FUNCTION_BLOCK FB_WindingControl
VAR_INPUT
	// Input hmi connection from MAIN
	hmiConnection   : POINTER TO FB_hmi_connection;   // HMI connection
	eventLogger     : POINTER TO FB_EventLogger;      // Event logger
	fileReadWrite   : POINTER TO FB_fileReadWrite;    // File read/write
END_VAR

VAR
	// Temporary testing vars

	// Function Blocks

	// CONTROL VARS
	desiredTension          : LREAL := 0;         // Desired tension
	desiredLinspeed         : LREAL := 0;         // Desired linear speed
	unwinding               : BOOL  := FALSE;     // Unwinding flag
	desiredTurnCountPickup  : DINT  := 0;         // Desired turn count for pickup
	
	// Exit conditions
	target_turn_count       : DINT  := 0;         // Target turn count

	// STATUS VARS
	state                   : INT   := 0;         // State for state machine
	cnt                     : UINT  := 0;         // PLC cycle counter
	eta                     : LREAL := 0;         // Time till completion in seconds
	etaFormattedString      : STRING(255);        // Formatted ETA in format ETA: M:S
	progressPercent         : LREAL := 0;         // Progress percentage (0 to 100) based on turn count

	// COIL MODELS (currently not used)
	// coil_model_base_Xcords : ARRAY[0..MAX_COIL_TYPE_COUNT] OF ARRAY[1..MAX_SIZE_COIL_MODEL] OF LREAL;
	// coil_model_base_Ycords : ARRAY[0..MAX_COIL_TYPE_COUNT] OF ARRAY[1..MAX_SIZE_COIL_MODEL] OF LREAL;

	// coil_model_rot_Xcords  : ARRAY[0..MAX_COIL_TYPE_COUNT] OF ARRAY[1..MAX_SIZE_COIL_MODEL] OF LREAL;
	// coil_model_rot_Ycords  : ARRAY[0..MAX_COIL_TYPE_COUNT] OF ARRAY[1..MAX_SIZE_COIL_MODEL] OF LREAL;

	// AXIS LIST
	payoff_axis_list        : ARRAY[1..GVL.MAX_PAYOFF_COUNT] OF FB_Axis;   // Payoff axis list
	pickup_axis_list        : ARRAY[1..GVL.MAX_PICKUP_COUNT] OF FB_Axis;   // Pickup axis list

	// MISC
	numOfEnabledPayoff      : INT := 0;           // Number of enabled payoffs
	tStart                  : TIME;               // Start time
	tEnd                    : TIME;               // End time
	tElapsed                : TIME;               // Elapsed time
	


END_VAR

VAR CONSTANT
	input_bounds            : input_bounds;       // Input bounds
	MAX_COIL_TYPE_COUNT     : INT := 1;           // Number of coil types (counts from 0)
	MAX_SIZE_COIL_MODEL     : INT := 1205;        // Maximum size of coil model
	TARGET_PICKUP_FORCE     : LREAL := 10;        // Target pickup force
	pi                      : LREAL := 4 * ATAN(1); // PI for math reasons (might be built-in but couldn't find it)
END_VAR

METHOD accelerating_tension : BOOL
VAR_INPUT
END_VAR

VAR
	i: INT;
	pickupLinspeed: LREAL;
	dist: LREAL;
	desiredVelocity: LREAL;
	adjustedVelocity: LREAL;
END_VAR
IF unwinding THEN
	//to do update with unwinding feature
	//seg fault to exit program :D remove when implmenting 
	i:=0;
	pickup_axis_list[i].acceleration:=0;
ELSE
	


	pickup_axis_list[1].torque:=desiredTension*	pickup_axis_list[1].getDistToAxis();
	
	//TO DO need to find what to set these to. 
	// to do . velo limits do not function how I thought they would need to ask beckhoff how they work.
	pickup_axis_list[1].velocityLimitLow:=(desiredLinspeed/pickup_axis_list[1].getDistToAxis())*57.29578;
	pickup_axis_list[1].velocityLimitHigh:=1000000 ;
	
	pickup_axis_list[1].setTorque();
	
	pickupLinspeed:=pickup_axis_list[1].AXIS.NcToPlc.ActVelo*	pickup_axis_list[1].getDistToAxis()/57.2957;
	
	
	
	FOR i:=1 TO GVL.MAX_PAYOFF_COUNT DO
		IF payoff_axis_list[i].enabled THEN
			//ASSUMING CONTINOUS UPDATE LIKE FUNCTION
			//TO DO figure out directions
			
			
			payoff_axis_list[i].setVelocity();
			dist:=payoff_axis_list[i].getDistToAxis();
			
			
			desiredVelocity:=(desiredLinspeed/dist)*57.29578;
			adjustedVelocity:=(pickupLinspeed/dist)*57.29578;
			
			
			//sets payoff axis to half way point between target linspeed and the actual linspeed.
			//i hope that this will give the pickup motor time to ramp up, while not giving too much speed to these motors.
			payoff_axis_list[i].velocity:=(desiredVelocity+adjustedVelocity)/2;
			
			
			
		END_IF
	END_FOR 
END_IF
END_METHOD

METHOD all_check : BOOL
VAR_INPUT
	write: BOOL;
END_VAR
all_check:= all_check OR general_input_check(write:=write);
all_check:= all_check OR payoff_input_check(write:=write);
all_check:=all_check OR pickup_input_check(write:=write);
END_METHOD

METHOD count_enabled_motors : BOOL
VAR_INPUT
END_VAR

VAR
	i: INT;
END_VAR
 //updates status of all axises, pickup and payoff

numOfEnabledPayoff:=0;

FOR i:= 1 TO GVL.MAX_PAYOFF_COUNT DO
IF	payoff_axis_list[i].enabled THEN
	numOfEnabledPayoff:=numOfEnabledPayoff+1;
END_IF
END_FOR
END_METHOD

METHOD CYCLIC : BOOL
VAR
	
	i: INT;
	

	intital: BOOL;
	errorOutput: BOOL;
	errorStatus: BOOL;
	
END_VAR
//cycle counter
cnt := cnt +1;

//-------------------------------------------------------------------------------------------------------------- USER INPUT --------------------------------------------------------------------------------------------------------------
	CASE state OF
		10:
		// ========================================10========================================
		IF hmiConnection^.resetUI THEN
		reset();
		hmiConnection^.resetUI:=FALSE;
		END_IF
	
		IF hmiConnection^.startUI THEN
			ADSLOGSTR(msgCtrlMask := ADSLOG_MSGTYPE_ERROR OR ADSLOG_MSGTYPE_MSGBOX,
				 msgFmtStr := 'Error Occured. Unable to start winding while not in tension state',
				 strArg:= '');
			hmiConnection^.startUI:=FALSE;
			
		END_IF
		IF hmiConnection^.tensionUI THEN
		state:=20;
		errorOutput:=TRUE;
		END_IF
	
		//check inputs button
		IF hmiConnection^.checkInputsUI THEN
			all_check(write:=FALSE);
			hmiConnection^.checkInputsUI:=FALSE;
			
		END_IF
		
		//update inputs button
		IF hmiConnection^.updateInputsUI THEN
			all_check(write:=TRUE);
			hmiConnection^.updateInputsUI:= FALSE;
			 
		END_IF
		
		IF hmiConnection^.homeUI THEN
			state:=50;
			errorOutput:=TRUE;
		END_IF
		
		IF hmiConnection^.estopHW THEN
			state:=500;

		END_IF
		
		
		// ========================================10========================================
		
		20,21:
		// ========================================20========================================
		
		//tension button
		IF hmiConnection^.resetUI THEN
		reset();
		hmiConnection^.resetUI:=FALSE;
		END_IF
	
		//start button
		IF hmiConnection^.startUI THEN
			state:=30;
			errorOutput:=TRUE;
		END_IF
		
		//tension button
		IF NOT hmiConnection^.tensionUI THEN
		state:=10;
		errorOutput:=TRUE;
		END_IF
	
		//check inputs button
		IF hmiConnection^.checkInputsUI THEN
			all_check(write:=FALSE);
			hmiConnection^.checkInputsUI:=FALSE;
		END_IF
		
		//update inputs button
		IF hmiConnection^.updateInputsUI THEN
			all_check(write:=TRUE);
			hmiConnection^.updateInputsUI:= FALSE;
			
		END_IF
		
		IF hmiConnection^.homeUI THEN
			ADSLOGSTR(msgCtrlMask := ADSLOG_MSGTYPE_ERROR OR ADSLOG_MSGTYPE_MSGBOX,
				 msgFmtStr := 'Error Occured. Unable to home outside of standby state',
				 strArg:= '');
			hmiConnection^.homeUI:=FALSE;
		END_IF
		
		IF hmiConnection^.estopHW THEN
			state:=500;

		END_IF
		
		// ========================================20========================================
		
		30,31,32,33:
		// ========================================30========================================
		
		//tension button
		IF hmiConnection^.resetUI THEN
			ADSLOGSTR(msgCtrlMask := ADSLOG_MSGTYPE_ERROR OR ADSLOG_MSGTYPE_MSGBOX,
				 msgFmtStr := 'Error Occured. Unable to reset during winding. Please pause winding.',
				 strArg:= '');
			hmiConnection^.resetUI:=FALSE;
			
		END_IF
	
		//start button
		IF NOT hmiConnection^.startUI THEN
			state:=20;
			errorOutput:=TRUE;
		END_IF
		
		//tension button
		IF NOT hmiConnection^.tensionUI THEN
			hmiConnection^.startUI:=FALSE;
			state:=10;
			errorOutput:=TRUE;
		END_IF
	
		//check inputs button
		IF hmiConnection^.checkInputsUI THEN
			all_check(write:=FALSE);
			hmiConnection^.checkInputsUI:=FALSE;
			errorOutput:=TRUE;
		END_IF
		
		//update inputs button
		IF hmiConnection^.updateInputsUI THEN
			all_check(write:=TRUE);
			hmiConnection^.updateInputsUI:=FALSE;
			
		END_IF
		
		IF hmiConnection^.homeUI THEN
			ADSLOGSTR(msgCtrlMask := ADSLOG_MSGTYPE_ERROR OR ADSLOG_MSGTYPE_MSGBOX,
				 msgFmtStr := 'Error Occured. Unable to home outside of standby state',
				 strArg:= '');
			hmiConnection^.homeUI:=FALSE;
		END_IF
		
		IF hmiConnection^.estopHW THEN
			state:=500;

		END_IF
		// ========================================30========================================
		
		
		40,41:
		// ========================================40========================================
		//tension button
		IF  hmiConnection^.tensionUI THEN
			state:=40;
			errorOutput:=TRUE;
		ELSE
			state:=41;
			
		END_IF
		
		//reset button
		IF hmiConnection^.resetUI THEN
			reset();
			hmiConnection^.resetUI:=FALSE;
			
		END_IF
	
		//start button
		IF hmiConnection^.startUI THEN
			ADSLOGSTR(msgCtrlMask := ADSLOG_MSGTYPE_ERROR OR ADSLOG_MSGTYPE_MSGBOX,
				 msgFmtStr := 'Error Occured. Unable to start while finished. Please reset first.',
				 strArg:= '');
			hmiConnection^.resetUI:=FALSE;
			
		END_IF
		
		//check inputs button
		IF hmiConnection^.checkInputsUI THEN
			all_check(write:=FALSE);
			hmiConnection^.checkInputsUI:=FALSE;
		END_IF
		
		//update inputs button
		IF hmiConnection^.updateInputsUI THEN
			all_check(write:=TRUE);
			hmiConnection^.updateInputsUI:= FALSE;
			
		END_IF
		
		IF hmiConnection^.homeUI THEN
			ADSLOGSTR(msgCtrlMask := ADSLOG_MSGTYPE_ERROR OR ADSLOG_MSGTYPE_MSGBOX,
				 msgFmtStr := 'Error Occured. Unable to home outside of standby state',
				 strArg:= '');
			hmiConnection^.homeUI:=FALSE;
		END_IF
		
		IF hmiConnection^.estopHW THEN
			state:=500;

		END_IF
		// ========================================40========================================

		// ========================================400========================================
		400:
			
		
		//reset button
		IF hmiConnection^.resetUI THEN
			reset();
			state:=10;
			hmiConnection^.resetUI:=FALSE;
			errorOutput:=TRUE;
		END_IF
	
		//start button
		IF hmiConnection^.startUI THEN
			ADSLOGSTR(msgCtrlMask := ADSLOG_MSGTYPE_ERROR OR ADSLOG_MSGTYPE_MSGBOX,
				 msgFmtStr := 'Error Occured. Unable to start while in error state. Please reset first, and resolve error.',
				 strArg:= '');
			hmiConnection^.resetUI:=FALSE;
			
		END_IF
		
		//check inputs button
		IF hmiConnection^.checkInputsUI THEN
			all_check(write:=FALSE);
			hmiConnection^.checkInputsUI:=FALSE;
		END_IF
		
		//update inputs button
		IF hmiConnection^.updateInputsUI THEN
			all_check(write:=TRUE);
			hmiConnection^.updateInputsUI:= FALSE;
			
		END_IF
		
		IF hmiConnection^.homeUI THEN
			ADSLOGSTR(msgCtrlMask := ADSLOG_MSGTYPE_ERROR OR ADSLOG_MSGTYPE_MSGBOX,
				 msgFmtStr := 'Error Occured. Unable to home inside error state. Please resolve errors on enabled axises',
				 strArg:= '');
			hmiConnection^.homeUI:=FALSE;
		END_IF
		
		IF hmiConnection^.estopHW THEN
			state:=500;

		END_IF
		// ========================================400========================================
		
		// =======================================50========================================
		50:
		IF  hmiConnection^.tensionUI THEN
				ADSLOGSTR(msgCtrlMask := ADSLOG_MSGTYPE_ERROR OR ADSLOG_MSGTYPE_MSGBOX,
				 msgFmtStr := 'Error Occured. Unable to tension while in homing sdtate. Please stop homing.',
				 strArg:= '');
			hmiConnection^.resetUI:=FALSE;
			
		END_IF
		
		//reset button
		IF hmiConnection^.resetUI THEN
			reset();
			state:=10;
			hmiConnection^.resetUI:=FALSE;
			errorOutput:=TRUE;
		END_IF
	
		//start button
		IF hmiConnection^.startUI THEN
			ADSLOGSTR(msgCtrlMask := ADSLOG_MSGTYPE_ERROR OR ADSLOG_MSGTYPE_MSGBOX,
				 msgFmtStr := 'Error Occured. Unable to start while in homing sdtate. Please stop homing.',
				 strArg:= '');
			hmiConnection^.resetUI:=FALSE;
			
		END_IF
		
		//check inputs button
		IF hmiConnection^.checkInputsUI THEN
			all_check(write:=FALSE);
			hmiConnection^.checkInputsUI:=FALSE;
		END_IF
		
		//update inputs button
		IF hmiConnection^.updateInputsUI THEN
			all_check(write:=TRUE);
			hmiConnection^.updateInputsUI:= FALSE;
			
		END_IF
		
		IF hmiConnection^.homeUI THEN
			
			hmiConnection^.homeUI:=FALSE;
			state:=10;
			errorOutput:=TRUE;
		END_IF
		
		IF hmiConnection^.estopHW THEN
			state:=500;

		END_IF
		// ========================================50========================================
		
		// =======================================500========================================
		500:
		IF  hmiConnection^.tensionUI THEN
				ADSLOGSTR(msgCtrlMask := ADSLOG_MSGTYPE_ERROR OR ADSLOG_MSGTYPE_MSGBOX,
				 msgFmtStr := 'Error Occured. Unable to tension while in ESTOP state. Please reset first.',
				 strArg:= '');
			hmiConnection^.tensionUI:=FALSE;
			
		END_IF
		
		//reset button
		IF hmiConnection^.resetUI THEN
			reset();
			state:=10;
			hmiConnection^.resetUI:=FALSE;
			errorOutput:=TRUE;
		END_IF
	
		//start button
		IF hmiConnection^.startUI THEN
			ADSLOGSTR(msgCtrlMask := ADSLOG_MSGTYPE_ERROR OR ADSLOG_MSGTYPE_MSGBOX,
				 msgFmtStr := 'Error Occured. Unable to start while in ESTOP state. Please reset first.',
				 strArg:= '');
			hmiConnection^.startUI:=FALSE;
			
		END_IF
		
		//check inputs button
		IF hmiConnection^.checkInputsUI THEN
			all_check(write:=FALSE);
			hmiConnection^.checkInputsUI:=FALSE;
		END_IF
		
		//update inputs button
		IF hmiConnection^.updateInputsUI THEN
			all_check(write:=TRUE);
			hmiConnection^.updateInputsUI:= FALSE;
			
		END_IF
		
		IF hmiConnection^.homeUI THEN
			ADSLOGSTR(msgCtrlMask := ADSLOG_MSGTYPE_ERROR OR ADSLOG_MSGTYPE_MSGBOX,
			msgFmtStr := 'Error Occured. Unable to home while in ESTOP state. Please reset first.',
			strArg:= '');
			hmiConnection^.homeUI:=FALSE;
		END_IF
		
		IF hmiConnection^.estopHW THEN
			state:=500;

		END_IF
		// ========================================500========================================
	END_CASE
//-------------------------------------------------------------------------------------------------------------- USER INPUT --------------------------------------------------------------------------------------------------------------
	
//clear status vars for axis. we will update them depending on our current state.
pickup_axis_list[1].setClear();

FOR i:= 1 TO GVL.MAX_PAYOFF_COUNT DO
	payoff_axis_list[i].setClear();
END_FOR

//check FOR error, IF error THEN set state TO 400

general_error_check(errorStatus=>errorStatus,errorOutput:=errorOutput);


//if no error, but currently in error state set winding to standby
//if none of the above state is unmodified
IF errorStatus THEN
	state:=400;
ELSIF state=400 AND NOT errorStatus THEN
	state:=10;
END_IF

//update HMI with certain motor values. 
hmi_update();



//-------------------------------------------------------------------------------------------------------------- MOTOR CONTROL --------------------------------------------------------------------------------------------------------------
CASE state OF
	00: //INIT STATE
	
	tstart:=TIME();
	state:=10;
	// ========================================10========================================
	10: //STANDBY STATE. 
	//wait for user inputs to transition to tension state. All motors are idle. Can edit params
	
	stop_all();
	// ========================================20========================================
	20: //STANDBY WITH STANDSTILL TENSION INITAL
	//inital error check for standstill tension state
	
	count_enabled_motors();
	//check inputs for standstill tension
	IF standstill_tension_check() THEN
		//if error then revert to standby
		state:=10;
		hmiConnection^.tensionUI:=FALSE;
	ELSE
		state:=21;
		
	END_IF
	// ========================================20========================================
	
	// ========================================21========================================
	21://STANDBY WITH STANDSTILL TENSION
	//no movement in cable, but tension is being created. waiting on user inputs to start winding. Can edit params
	
	
	standstill_tension();
	// ========================================21========================================

	// ========================================30========================================
	30: //WINDING TENSION INITAL
	//inital error check for winding tension state.
	
	count_enabled_motors();
	// INPUT VALIDATION
	IF winding_check() THEN
		//if error then revert to standby
		state:=20;
		hmiConnection^.startUI:=FALSE;
		
		
		
	ELSE
		eventLogger^.fbMessage[1].Send(0);
		state:=31;
		tStart:=TIME();
	END_IF
	// ========================================30========================================
	
	// ========================================31========================================
	31: //WINDING TENSION, ACCELERATION
	//coil is currently ramping speed. can not edit params.
	
	

	
	accelerating_tension();
	determine_motor_state();
	tElapsed:=TIME() -tStart;
	
	IF winding_exit_check() THEN
	
		state:=39;
		
	ELSE
		state:=31;
	END_IF
	
	
	// ========================================31========================================
	
	// ========================================32========================================
	32: //WINDING TENSION, STEADY STATE
	//coil is in steady state. moving at constant velo with set tension. Can not edit params
	
	
	
	winding_tension();
	determine_motor_state();
	tElapsed:=TIME() -tStart;

	//check for exit conditions 
	IF winding_exit_check() THEN
		
		state:=39;
		
	ELSE
		state:=32;
	END_IF
	
	
	
	// ========================================32========================================
	
	// ========================================33========================================
	33: //WINDING TENSION, DEACCELERATION
	//coil currently decreasing speed, while maintaining. Can not edit params
	

	
	decelerating_tension();
	determine_motor_state();
	tElapsed:=TIME() -tStart;

	//check for exit conditions 
	IF winding_exit_check() THEN
		
		state:=39;
		
	ELSE
		state:=33;
	END_IF
	// ========================================33========================================
	
	// ========================================39========================================
	39: // transition state from winding => finished
		eventLogger^.fbMessage[2].Send(0);
		hmiConnection^.startUI:=FALSE;
		
		tEnd:=TIME();
		tElapsed:=tEnd -Tstart;
		
		fileReadWrite^.update_database(user:= 'RN',
										timeStarted:=tStart,
										timeCompleted:=tEnd,
										timeElasped:=tElapsed,
										numOfCoil:=numOfEnabledPayoff,
										lengthOCoil:=numOfEnabledPayoff,
										userNote:='TO DO need to add user logging feature');
		fileReadWrite^.bWrite:=TRUE;			
		
	
		state:=40;
	// ========================================39========================================
	
	
	// ========================================40========================================
	40: //FINISHED HOLD STANDSTILL TENSION
	//cable winding finished, currently mainting tension until user input. Can not edit params
	
	standstill_tension();
	
	IF standstill_tension_check() THEN
		//if error then revert to standby
		state:=51;
		
	ELSE
		state:=40;
		
	END_IF
	// ========================================40========================================
	
	// ========================================41========================================
	41: //FINISHED NO TENSION
	//cable winding finished, waiting on user reset to transition to standby state. Can edit params
	//do not control tension
	
	// ========================================41========================================
	

	// ========================================50========================================
	50:
	//exit homing state if homing is done or error.
	IF set_pos_all() THEN
		state:=10;
		hmiConnection^.homeUI:=FALSE;
	
	ELSE
		state:=50;
	END_IF
	
	
	
	
	
	// ========================================50========================================
	
	// ========================================51========================================
	
	400: //ERROR STATE
	//error on a axis preventing motor movement, or winding start. //do nothing 'till resolved
	500: //ESTOP STATE
	//triggered on estop press. can be cleared with reset
		estop_routine();
		
	
END_CASE
//-------------------------------------------------------------------------------------------------------------- MOTOR CONTROL --------------------------------------------------------------------------------------------------------------

//get status updates
//only calculate once very N turns in order to save resources. there also shouldnt be need to run eveyr plc cycle
	
IF (cnt MOD 10 =0) and  NOT(desiredLinspeed = 0) THEN
	etaFormattedString:=find_eta();
	progressPercent :=get_current_progress();
END_IF


//Call cyclic methods of all axies 
pickup_axis_list[1].CYLIC();

FOR i:= 1 TO GVL.MAX_PAYOFF_COUNT DO
	payoff_axis_list[i].CYLIC();
END_FOR
END_METHOD

METHOD decelerating_tension : BOOL
VAR_INPUT
END_VAR
END_METHOD

METHOD determine_motor_state : BOOL
VAR_INPUT
END_VAR





VAR
	actualLinspeed : LREAL;
END_VAR
//to do . comeback on this and do a once over. not sure if this is what we want.
			
actualLinspeed:=pickup_axis_list[1].getDistToAxis()*pickup_axis_list[1].actualVelocity/57.29578;
		
//if we are below our desired
IF actualLinspeed <= 0.9*desiredLinspeed THEN
	
	state:=31;

//last turn dedicated to decelerating 
ELSIF pickup_axis_list[1].AXIS.NcToPlc.ModuloActTurns = desiredTurnCountPickup-1 THEN

	state:=33;

//if not accelerating or decelerating then we are in steady state
ELSE

	state:=32;
	
END_IF
END_METHOD

METHOD estop_routine : BOOL
VAR_INPUT
END_VAR

VAR
	i: INT;
END_VAR
//during estop, cut power to motors.

//turn power off on all axies. 
pickup_axis_list[1].MCPOWER(Axis:=pickup_axis_list[1].AXIS,ENABLE:=FALSE);

FOR i:=1 TO GVL.MAX_PAYOFF_COUNT DO
		payoff_axis_list[i].MCPOWER(Axis:=payoff_axis_list[i].AXIS,ENABLE:=FALSE);
END_FOR
END_METHOD

//updates eta var
METHOD find_eta : STRING(255)
VAR
	length : LREAL; //length of straight sections in race track coil
	minutes: DINT;
	
	seconds: DINT;
	minutesString: STRING;
	secondsString: STRING;
	formattedString: STRING(255);
	tape_thicnes: LREAL :=0; //total tape thickness in meters
	i: INT;
	total_circum: LREAL;
	currentTurnCount: LREAL;
	currentCircum: LREAL;
END_VAR
VAR CONSTANT
	pi : LREAL := 4 * ATAN(1);
END_VAR
//if we are finished out put 0 seconds and exit
IF state <=59 AND state >= 50 THEN
eta:=0;
RETURN ;
END_IF

CASE pickup_axis_list[1].coilShapeID OF
	//finds eta given turn count
	//formulas are a function of circumfrence given turn count. we take the intergral of this, with respect to turn count, with the upper bound being our target turn count 
	0:
	
	tape_thicnes:=0;
	FOR i:=1 TO GVL.MAX_PAYOFF_COUNT DO
		IF payoff_axis_list[i].enabled THEN
		tape_thicnes:=tape_thicnes+payoff_axis_list[i].tape_info[payoff_axis_list[i].tapeType].tape_depth/1000;
		END_IF
	END_FOR
	

	
	
	
	total_circum:=2*pi*desiredTurnCountPickup*pickup_axis_list[1].pancake.radius/1000 + tape_thicnes*EXPT(desiredTurnCountPickup,2)*pi;
	
	currentTurnCount:=pickup_axis_list[1].AXIS.NcToPlc.ModuloActPos/360+pickup_axis_list[1].AXIS.NcToPlc.ModuloActTurns;
	
	currentCircum:=2*pi*currentTurnCount*pickup_axis_list[1].pancake.radius/1000 +tape_thicnes*EXPT(currentTurnCount,2)*pi;
	
	IF NOT(desiredLinspeed =0) THEN
		eta:=(total_circum-currentCircum)/desiredLinspeed;
	ELSE
		eta:=0;
	END_IF
	

	
	
	
	1:	
	// to do. update this monster of a formula for the race track coil. derived through calculus, which is probably correct, just now cant figure it out because i decided to write a one liner instead of splitting up
	(*
	eta:=((2*pi*racetrack_params.radius*target_turn_count_pickup+pi*tape_info.tape_depth*target_turn_count_pickup*target_turn_count_pickup+2*racetrack_params.length*target_turn_count_pickup)
		 -(2*pi*racetrack_params.radius*pickup_motor_list[1].turn_count+pi*tape_info.tape_depth*target_turn_count_pickup*pickup_motor_list[1].turn_count+2*racetrack_params.length*pickup_motor_list[1].turn_count));
		 *)
END_CASE


// Convert the LREAL value to minutes and seconds
minutes := TRUNC(eta / 60);
seconds := TRUNC(eta - (minutes * 60));

// Convert the minutes and seconds to strings
minutesString := DINT_TO_STRING(minutes);
secondsString := DINT_TO_STRING(seconds);

// Format the final output string
find_eta := CONCAT(CONCAT('ETA: ', minutesString), CONCAT(':', secondsString));
END_METHOD

METHOD general_error_check : BOOL
VAR
	i: INT;
	pickup_motor_count: INT;
	adsError : BOOL;
END_VAR
VAR_OUTPUT
	errorStatus : BOOL ;
END_VAR
VAR_IN_OUT
	errorOutput: BOOL ;
END_VAR
//Checks to see if there are any errors in a enabled axis.


pickup_axis_list[1].error_check_all();

errorStatus:=pickup_axis_list[1].AXIS.Status.Error OR pickup_axis_list[1].adsError ;
		
IF errorOutput AND pickup_axis_list[1].AXIS.Status.Error THEN
			
			ADSLOGSTR(
        		msgCtrlMask := ADSLOG_MSGTYPE_ERROR OR ADSLOG_MSGTYPE_MSGBOX,
        		msgFmtStr := 'Error occurred. Error on Pickup Axis with ID: %S',
        		strArg := UDINT_TO_STRING(pickup_axis_list[1].AXIS.Status.ErrorID)
   			 );
		
			errorOutput:=FALSE;
		
END_IF
		
IF errorOutput AND pickup_axis_list[1].adsError THEN
			
			ADSLOGSTR(
        		msgCtrlMask := ADSLOG_MSGTYPE_ERROR OR ADSLOG_MSGTYPE_MSGBOX,
        		msgFmtStr := 'Error occurred. Error in Pickup Axis FB with ID: %S ',
        		strArg := UDINT_TO_STRING(pickup_axis_list[1].adsErrorID)
   			 );
		
			errorOutput:=FALSE;
		
END_IF



FOR i:= 1 TO GVL.MAX_PAYOFF_COUNT DO
	
	payoff_axis_list[i].error_check_all();

	
		errorStatus:=errorStatus OR ((payoff_axis_list[i].AXIS.Status.Error OR payoff_axis_list[i].adsError) AND payoff_axis_list[i].enabled);
		
		IF errorOutput AND payoff_axis_list[i].AXIS.Status.Error THEN
			
			ADSLOGSTR(
        		msgCtrlMask := ADSLOG_MSGTYPE_ERROR OR ADSLOG_MSGTYPE_MSGBOX,
        		msgFmtStr := 'Error occurred. Error on Pickup Axis with ID: %S',
        		strArg := UDINT_TO_STRING(payoff_axis_list[i].AXIS.Status.ErrorID)
   			 );
		
			errorOutput:=FALSE;
		
END_IF
		
IF errorOutput AND payoff_axis_list[i].adsError THEN
			
			ADSLOGSTR(
        		msgCtrlMask := ADSLOG_MSGTYPE_ERROR OR ADSLOG_MSGTYPE_MSGBOX,
        		msgFmtStr := 'Error occurred. Error in Pickup Axis FB with ID: %S ',
        		strArg := UDINT_TO_STRING(payoff_axis_list[i].adsErrorID)
   			 );
		
			errorOutput:=FALSE;
		
END_IF
		
END_FOR
END_METHOD

METHOD general_input_check : BOOL
VAR_INPUT
	write: BOOL;
END_VAR
IF hmiConnection^.general_input_datagrid_params_list[1].tension < input_bounds.tension_low OR hmiConnection^.general_input_datagrid_params_list[1].tension > input_bounds.tension_high THEN
	general_input_check := TRUE;
	
	ADSLOGSTR(
        	msgCtrlMask := ADSLOG_MSGTYPE_ERROR OR ADSLOG_MSGTYPE_MSGBOX,
        	msgFmtStr := 'Error occurred. Tension outside of range. ',
        	strArg := ''
   		 );
	
ELSE
	
	IF write THEN
		desiredTension:=hmiConnection^.general_input_datagrid_params_list[1].tension;
	
	END_IF
END_IF

IF hmiConnection^.general_input_datagrid_params_list[1].linspeed < input_bounds.linear_speed_low OR hmiConnection^.general_input_datagrid_params_list[1].linspeed > input_bounds.linear_speed_high THEN
	general_input_check := TRUE;
	
	ADSLOGSTR(
        	msgCtrlMask := ADSLOG_MSGTYPE_ERROR OR ADSLOG_MSGTYPE_MSGBOX,
        	msgFmtStr := 'Error occurred. Linear speedc out of range.',
        	strArg := ''
   		 );
	
ELSE
	IF write THEN
		desiredLinspeed:=hmiConnection^.general_input_datagrid_params_list[1].linspeed;
	
	END_IF
	
END_IF

IF write THEN
	unwinding:=hmiConnection^.general_input_datagrid_params_list[1].unwinding;
	
END_IF
END_METHOD

METHOD get_current_progress : LREAL
IF unwinding THEN
	get_current_progress := 100-(pickup_axis_list[1].AXIS.NcToPlc.ModuloActTurns/desiredTurnCountPickup)*100;
	
ELSE
	get_current_progress := ((pickup_axis_list[1].AXIS.NcToPlc.ModuloActPos/360+pickup_axis_list[1].AXIS.NcToPlc.ModuloActTurns)/desiredTurnCountPickup)*100;

END_IF
END_METHOD

METHOD hmi_update : BOOL
VAR_INPUT
END_VAR

VAR
	i: INT;
END_VAR
//collection of functions to update hmi vars. 

hmiConnection^.state:=state;

update_error_status();
update_torque();
update_velocity();



hmiConnection^.overview_outputs_datagrid_list[1].pickupTurnCount:=pickup_axis_list[1].AXIS.NcToPlc.ModuloActPos/360+pickup_axis_list[1].AXIS.NcToPlc.ModuloActTurns;
hmiConnection^.overview_outputs_datagrid_list[1].linspeed:=pickup_axis_list[1].actualVelocity*payoff_axis_list[1].getDistToAxis()/57.29578;
hmiConnection^.overview_outputs_datagrid_list[1].torque:=pickup_axis_list[1].actualTorque/pickup_axis_list[1].getDistToAxis();

hmiConnection^.turncount_output_datagrid_list[1].pickupTC1:=pickup_axis_list[1].AXIS.NcToPlc.ModuloActPos/360+pickup_axis_list[1].AXIS.NcToPlc.ModuloActTurns;
hmiConnection^.turncount_output_datagrid_list[1].payoffTC1:=payoff_axis_list[1].AXIS.NcToPlc.ModuloActPos/360+payoff_axis_list[1].AXIS.NcToPlc.ModuloActTurns;
hmiConnection^.turncount_output_datagrid_list[1].payoffTC2:=payoff_axis_list[2].AXIS.NcToPlc.ModuloActPos/360+payoff_axis_list[2].AXIS.NcToPlc.ModuloActTurns;
hmiConnection^.turncount_output_datagrid_list[1].payoffTC3:=payoff_axis_list[3].AXIS.NcToPlc.ModuloActPos/360+payoff_axis_list[3].AXIS.NcToPlc.ModuloActTurns;
END_METHOD

METHOD home : BOOL
VAR_INPUT
END_VAR

VAR
	i: INT;
END_VAR
//to do . something about the set pos function is broken but not sure what. in duplicate project i was able to replicate the error so either 
//it is something to do with virtual axis, or bug in twincat. may need to find workaround with drive manager. 


//check to see if we are done
pickup_axis_list[1].setPos();
home := home AND pickup_axis_list[1].MCPOS.Done ;
	

	FOR i:=1 TO GVL.MAX_PAYOFF_COUNT DO
		IF payoff_axis_list[i].enabled THEN
			payoff_axis_list[i].setPos();
			home := home AND payoff_axis_list[i].MCPOS.Done ;
		END_IF
			
	END_FOR

	
//cancels home if we run into any error
//home := home OR pickup_axis_list[1].MCPOS.Error;
	
FOR i:=1 TO GVL.MAX_PAYOFF_COUNT DO
	IF payoff_axis_list[i].enabled THEN
		
		payoff_axis_list[i].setPos();
		home := home AND payoff_axis_list[i].MCPOS.Done;
	END_IF
			
END_FOR
END_METHOD

METHOD INIT : BOOL
VAR_INPUT
END_VAR

VAR
	i: INT;
END_VAR
init_coil_model();
//Call cyclic methods of all axies 

pickup_axis_list[1].INIT();

pickup_axis_list[1].torqaueConstrant:=GVL.PICKUP_TORQUE_CONSTANT;
pickup_axis_list[1].ratedCurrent:=GVL.PICKUP_RATED_CURRENT;
pickup_axis_list[1].enabled:=TRUE;

pickup_axis_list[1].gearRatioNum:=10;
pickup_axis_list[1].gearRatioDen:=1;
FOR i:= 1 TO GVL.MAX_PAYOFF_COUNT DO
	payoff_axis_list[i].INIT();
	payoff_axis_list[i].torqaueConstrant:=GVL.PAYOFF_TORQUE_CONSTANT;
	payoff_axis_list[i].ratedCurrent:=GVL.PAYOFF_RATED_CURRENT;
	payoff_axis_list[i].gearRatioNum:=60;
	payoff_axis_list[i].gearRatioDen:=1;
END_FOR

etaFormattedString := CONCAT(CONCAT('ETA: ', '0'), CONCAT(':', '0'));
END_METHOD

METHOD init_coil_model : BOOL
VAR 
	med_val : LREAL; // intermediate value 
	i :INT ;
	
	coil_type: INT:=0;
	cnt: INT :=0; //temp
END_VAR
VAR CONSTANT
	
END_VAR
//TO DO this funciton was orginall made to create a model of a non circular pickup coil shape. i would like to redo it. 

(*



	//1:
	//creates 1205 points to model a race track coil. we do this 
	cnt:=0;
	FOR i := -150 TO 150 DO
    	coil_model_base_Xcords[1][i+151]:=racetrack_params_1.radius+pickup_motor_list[1].turn_count*tape_info.tape_depth;
		coil_model_base_Ycords[1][i+151]:=i;
		
		
	END_FOR;
	FOR i := -150 TO 150 DO
    	coil_model_base_Xcords[1][i+452]:=-(coil_shape_params.radius+pickup_motor_list[1].turn_count*tape_info.tape_depth);
		coil_model_base_Ycords[1][i+452]:=i;
	
	END_FOR;
	FOR i := -150 TO 150 DO
		med_val:=(pi/300)*i+pi;
		
		
    	coil_model_base_Xcords[1][i+753]:=(coil_shape_params.radius+pickup_motor_list[1].turn_count*tape_info.tape_depth)*SIN(med_val);
		coil_model_base_Ycords[1][i+753]:=-1*coil_shape_params.length*COS(med_val);
	
	END_FOR;
	FOR i := -150 TO 150 DO
		med_val:=(pi/300)*i;
		
		
    	coil_model_base_Xcords[1][i+904]:=(coil_shape_params.radius+pickup_motor_list[1].turn_count*tape_info.tape_depth)*SIN(med_val);
		coil_model_base_Ycords[1][i+904]:=coil_shape_params.length*COS(med_val);
	
	END_FOR;
	 
*)
END_METHOD

METHOD input_update : BOOL
VAR_INPUT
	general : BOOL ;
	pickup : BOOL ;
	payoff : BOOL ;
END_VAR



VAR
	
	//chooses which inputs we will update.         
	i: INT;
END_VAR
//NOT NEEDED ANYMORE
(*


//Updates internal winding control variables with HMI inputs. 
IF pickup THEN
	pickup_axis_list[1].coilShapeID:=hmiConnection^.pickup_input_datagrid_params_list[1].coil_shape;
	desiredTurnCountPickup:=hmiConnection^.pickup_input_datagrid_params_list[1].turn_count;
END_IF

IF payoff THEN
	FOR i:= 1 TO GVL.MAX_PAYOFF_COUNT DO
		payoff_axis_list[i].enabled:=hmiConnection^.payoff_input_datagrid_params_list[i].enabled;
	IF payoff_axis_list[i].enabled THEN
		payoff_axis_list[i].pancake.radius:=hmiConnection^.payoff_input_datagrid_params_list[i].outer_dia;
		
	
	END_IF
	
	END_FOR
END_IF

IF general THEN
	desiredLinspeed:=hmiConnection^.general_input_datagrid_params_list[1].linspeed;
	desiredTension:=hmiConnection^.general_input_datagrid_params_list[1].tension;
	unwinding:=hmiConnection^.general_input_datagrid_params_list[1].unwinding;
	
	pickup_axis_list[1].directionB:=BOOL_TO_INT(unwinding);
	
	FOR i:= 1 TO GVL.MAX_PAYOFF_COUNT DO
		payoff_axis_list[i].directionB:=BOOL_TO_INT(unwinding);

	END_FOR
END_IF

*)
END_METHOD

METHOD payoff_input_check : BOOL
VAR_INPUT
END_VAR

VAR_input
	write: BOOL;
END_VAR
VAR
	i: INT;
END_VAR
 FOR i:= 1 TO GVL.MAX_PAYOFF_COUNT DO
	
	IF write THEN
		payoff_axis_list[i].enabled:=hmiConnection^.payoff_input_datagrid_params_list[i].enabled;
		payoff_axis_list[i].tapeType:=hmiConnection^.payoff_input_datagrid_params_list[i].tape_type;
	END_IF

	IF hmiConnection^.payoff_input_datagrid_params_list[i].enabled THEN
		
	
		IF hmiConnection^.payoff_input_datagrid_params_list[i].radius < input_bounds.radius_payoff_low OR hmiConnection^.payoff_input_datagrid_params_list[i].radius > input_bounds.radius_payoff_high THEN
		payoff_input_check := TRUE;
	
		ADSLOGSTR(
        	msgCtrlMask := ADSLOG_MSGTYPE_ERROR OR ADSLOG_MSGTYPE_MSGBOX,
        	msgFmtStr := 'Error occurred. Payoff Radius outside of range.',
        	strArg := ''
   		 );
		
		ELSE 
			IF write THEN
				payoff_axis_list[i].pancake.radius:=hmiConnection^.payoff_input_datagrid_params_list[i].radius;
			END_IF
		END_IF
	
	END_IF
	
END_FOR
END_METHOD

METHOD pickup_input_check : BOOL
VAR_INPUT
	write : BOOL ;
END_VAR
IF hmiConnection^.pickup_input_datagrid_params_list[1].turn_count < input_bounds.turn_count_pickup_low OR hmiConnection^.pickup_input_datagrid_params_list[1].turn_count > input_bounds.turn_count_pickup_high THEN
	pickup_input_check := TRUE;
	
	ADSLOGSTR(
        	msgCtrlMask := ADSLOG_MSGTYPE_ERROR OR ADSLOG_MSGTYPE_MSGBOX,
        	msgFmtStr := 'Error occurred. Pickup turncount outside of range.',
        	strArg := ''
   		 );
	
ELSE
	
	IF write THEN
		desiredTurnCountPickup:=hmiConnection^.pickup_input_datagrid_params_list[1].turn_count;
	END_IF

	
	
	
END_IF
END_METHOD

METHOD read_status : BOOL
VAR_INPUT
END_VAR

VAR
	i: INT;
END_VAR
 //updates status of all axises, pickup and payoff

pickup_axis_list[1].Axis.ReadStatus();


FOR i:= 1 TO GVL.MAX_PAYOFF_COUNT DO
	payoff_axis_list[i].AXIS.ReadStatus();
END_FOR
END_METHOD

METHOD reset : BOOL
VAR_INPUT
END_VAR
state := 10;
progressPercent:=0;
//TO DO . need to find out out to clear position to 0
END_METHOD

METHOD set_pos_all : BOOL
VAR_INPUT
END_VAR

VAR

	i: INT;
	busy : BOOL :=FALSE;
	busytemp : BOOL := FALSE;
	error : BOOL:= FALSE;
	errorTemp : BOOL := FALSE;
END_VAR
//to do . bug where after a failed winding attemp, users need to press button one more time inorder for command to run. coming back to this later

//function to set pos of all motors to 0

//turn power off on all axies. need for set pos function
pickup_axis_list[1].MCPOWER(Axis:=pickup_axis_list[1].AXIS,ENABLE:=FALSE);

FOR i:=1 TO GVL.MAX_PAYOFF_COUNT DO
	IF payoff_axis_list[i].enabled THEN
			
		payoff_axis_list[i].MCPOWER(Axis:=payoff_axis_list[i].AXIS,ENABLE:=FALSE);
	END_IF
END_FOR 




//set pos, repeat till not busy. 
REPEAT
	
	//set pos of pickup
	pickup_axis_list[1].MCPOS(Axis:=pickup_axis_list[1].Axis,Execute:=TRUE,Position:=0,MODE:=FALSE,busy=>busytemp,Error=>errortemp);
	busy:= busy AND busytemp;
	error:= error AND errorTemp;


//set pos of payoff
	FOR i:=1 TO GVL.MAX_PAYOFF_COUNT DO
		IF payoff_axis_list[i].enabled THEN
			
			payoff_axis_list[1].MCPOS(Axis:=payoff_axis_list[1].Axis,Execute:=TRUE,Position:=0,MODE:=FALSE,busy=>busytemp,Error=>errortemp);
			busy:=busy AND busytemp;
			error:= error AND errorTemp;
		END_IF
	END_FOR 


//exit condition	
UNTIL 
//exit when all axies are no longer busy
NOT BUSY
END_REPEAT

pickup_axis_list[1].MCPOS(Axis:=pickup_axis_list[1].Axis, Execute:=TRUE,Position:=0,mode:=FALSE);


set_pos_all:=TRUE;

//turn power off on all axies. 
pickup_axis_list[1].MCPOWER(Axis:=pickup_axis_list[1].AXIS,ENABLE:=TRUE);
pickup_axis_list[1].MCPOS(Axis:=pickup_axis_list[1].Axis,Execute:=FALSE,Position:=0,MODE:=FALSE,busy=>busytemp,Error=>errortemp);

FOR i:=1 TO GVL.MAX_PAYOFF_COUNT DO
	IF payoff_axis_list[i].enabled THEN
		payoff_axis_list[i].MCPOWER(Axis:=payoff_axis_list[i].AXIS,ENABLE:=TRUE);
		payoff_axis_list[i].MCPOS(Axis:=payoff_axis_list[1].Axis,Execute:=FALSE,Position:=0,MODE:=FALSE,busy=>busytemp,Error=>errortemp);
	END_IF		
END_FOR
END_METHOD

METHOD standstill_tension : BOOL
VAR_INPUT
END_VAR

VAR
	i: INT;
END_VAR
//creates tension in tape, but does not move the tape.

//set torque to force times number of payoff motors enabled. 
pickup_axis_list[1].torque:=(desiredTension*numOfEnabledPayoff*	pickup_axis_list[1].getDistToAxis())/2;
	
//TO DO need to find what to set these to. might be too low. 
pickup_axis_list[1].velocityLimitLow:=0;
pickup_axis_list[1].velocityLimitHigh:=1;
	
	
pickup_axis_list[1].setTorque();
	
	
FOR i:=1 TO GVL.MAX_PAYOFF_COUNT DO
	IF payoff_axis_list[i].enabled THEN
		payoff_axis_list[i].setTorque();
		
		payoff_axis_list[1].velocityLimitLow:=0;
		payoff_axis_list[1].velocityLimitHigh:=1;
		payoff_axis_list[i].torque:=-1*desiredTension*	payoff_axis_list[1].getDistToAxis()/2;
			
	END_IF
END_FOR
END_METHOD

METHOD standstill_tension_check : BOOL
VAR_OUTPUT

END_VAR
VAR
	input_bounds : input_bounds; //struct defining input bounds
	i: INT; //counter
	
	
	payoffEnableCheck :BOOL :=FALSE; //var to hold payoff enable var
END_VAR
//check to see if HMI vars are valid for stand still tension before winding. outputs true if there was an error.

//PICKUP AXIS CHECKS

IF hmiConnection^.general_input_datagrid_params_list[1].tension < input_bounds.tension_low OR hmiConnection^.general_input_datagrid_params_list[1].tension > input_bounds.tension_high THEN
	standstill_tension_check := TRUE;
	
	ADSLOGSTR(
        	msgCtrlMask := ADSLOG_MSGTYPE_ERROR OR ADSLOG_MSGTYPE_MSGBOX,
        	msgFmtStr := 'Error occurred. Tension outside of range. Unable to start tension',
        	strArg := ''
   		 );
	
ELSE
	desiredTension:=hmiConnection^.general_input_datagrid_params_list[1].tension;
	
END_IF

//PAYOFF AXIS CHECKS

FOR i:= 1 TO GVL.MAX_PAYOFF_COUNT DO
	payoffEnableCheck:=payoffEnableCheck OR hmiConnection^.payoff_input_datagrid_params_list[i].enabled;
	
END_FOR


IF NOT payoffEnableCheck THEN
	standstill_tension_check := TRUE;
	
	ADSLOGSTR(
        	msgCtrlMask := ADSLOG_MSGTYPE_ERROR OR ADSLOG_MSGTYPE_MSGBOX,
        	msgFmtStr := 'Error occurred. At least one payoff motor needs to be enabled',
        	strArg := ''
   		 );

END_IF
END_METHOD

METHOD stop_all : BOOL
VAR_INPUT
END_VAR

VAR
	i: INT;
END_VAR

	pickup_axis_list[1].setStop();
		
	FOR i:=1 TO GVL.MAX_PAYOFF_COUNT DO
		
			payoff_axis_list[i].setStop();
			
		
	END_FOR
END_METHOD

METHOD update_error_status : BOOL
VAR_INPUT
END_VAR

VAR
	i: INT;
	
END_VAR
hmiConnection^.output_error_datagrid_list[0].errorStatus:=pickup_axis_list[1].AXIS.Status.Error;
hmiConnection^.output_error_datagrid_list[0].errorID:=pickup_axis_list[1].AXIS.Status.ErrorID;

hmiConnection^.motor_state_datagrid_list[0].state:=pickup_axis_list[1].state;

FOR i:= 1 TO GVL.MAX_PAYOFF_COUNT DO
	hmiConnection^.output_error_datagrid_list[i].errorStatus:=payoff_axis_list[i].AXIS.Status.Error;
	hmiConnection^.output_error_datagrid_list[i].errorID:=payoff_axis_list[i].AXIS.Status.ErrorID;
	
	hmiConnection^.motor_state_datagrid_list[i].state:=payoff_axis_list[i].state;
	
END_FOR
END_METHOD

METHOD update_torque : BOOL
VAR_INPUT
END_VAR

VAR
	i: INT;
END_VAR
//update act ual torque values ofc motors. send these values to HMI

pickup_axis_list[1].getTorque();
hmiConnection^.torque[1]:=pickup_axis_list[1].actualTorque;


FOR i:= 1 TO GVL.MAX_PAYOFF_COUNT DO
	payoff_axis_list[i].getTorque();
	hmiConnection^.torque[i+1]:=payoff_axis_list[i].actualTorque;

END_FOR
END_METHOD

METHOD update_velocity : BOOL
VAR_INPUT
END_VAR

VAR
	i: INT;
END_VAR
//update act ual torque values ofc motors. send these values to HMI


hmiConnection^.rpm[1]:=pickup_axis_list[1].actualVelocity;


FOR i:= 1 TO GVL.MAX_PAYOFF_COUNT DO

	hmiConnection^.rpm[i+1]:=payoff_axis_list[i].actualVelocity;

END_FOR
END_METHOD

METHOD winding_check : BOOL
VAR_INPUT
END_VAR
END_METHOD

METHOD winding_exit_check : BOOL
VAR_INPUT
END_VAR
//Checks to see if various conditions are met to exit

//turn count condition.

IF pickup_axis_list[1].AXIS.NcToPlc.ModuloActTurns >= desiredTurnCountPickup THEN
	winding_exit_check :=TRUE;
		
	ADSLOGSTR(msgCtrlMask := ADSLOG_MSGTYPE_HINT OR ADSLOG_MSGTYPE_MSGBOX, msgFmtStr := 'Winding stopped, pickup turn count reached', strArg:= '');
END_IF
END_METHOD

METHOD winding_tension : BOOL
VAR_INPUT
END_VAR

VAR
	i: INT;
	
	desiredVelocity : LREAL;
	pickupLinspeed: LREAL;
	adjustedVelocity: LREAL;
	dist: LREAL;
END_VAR
VAR CONSTANT
	PERCENT_DIFFERENCE: LREAL := 1.1;
END_VAR
IF unwinding THEN
	//to do update with unwinding feature
	
	//do nothing, not implemneted yet. 
ELSE
	


	pickup_axis_list[1].torque:=desiredTension*numOfEnabledPayoff*	pickup_axis_list[1].getDistToAxis();
	
	//TO DO . need to confirm these are correct
	//how i envison the limits to function is that the pickup side will gradually ramp up speed until we hit the upper velocity limit. we could maybe have no limits and just have only torque control
	//will need testing. 
	pickup_axis_list[1].velocityLimitLow:=0;
	pickup_axis_list[1].velocityLimitHigh:=(desiredLinspeed/pickup_axis_list[1].getDistToAxis())*57.29578 ;
	
	pickup_axis_list[1].setTorque();
	
	pickupLinspeed:=pickup_axis_list[1].AXIS.NcToPlc.ActVelo*	pickup_axis_list[1].getDistToAxis()/57.2957;
	
	
	
	FOR i:=1 TO GVL.MAX_PAYOFF_COUNT DO
		IF payoff_axis_list[i].enabled THEN
			//ASSUMING CONTINOUS UPDATE LIKE FUNCTION
			//TO DO figure out directions
			
			
			payoff_axis_list[i].setVelocity();
			dist:=payoff_axis_list[i].getDistToAxis();
			
			//find the velocity (degree/s) to acheive our desired linear speed, and the linear speed at pickup motor. 
			desiredVelocity:=(desiredLinspeed/dist)*57.29578;
			adjustedVelocity:=(pickupLinspeed/dist)*57.29578;
			
			
			//sets payoff axis to half way point between target linspeed and the actual linspeed.
			//how i envison this to function, is that while pickup side is at a low speed, the payoff side will also work at a lower speed,
			//which gives the pickup time to catch up in speed. right now i do this by just averaging desired speed and actual speed,
			//this could maybe he handled in a better way, so i will leave a TO DO 
			payoff_axis_list[i].velocity:=(desiredVelocity+adjustedVelocity)/2;
			
			
			
		END_IF
	END_FOR 
END_IF
END_METHOD

END_FUNCTION_BLOCK

(* stored: Version 1.1.0.1, ProductVersion 3.1.4024.12
   POU FB_WindingControl: Id {2bf4d53e-3c0a-48b3-b562-160f25601b83}, SpecialFunc None
   Folder Methods: Id {b393cdcb-7058-41c2-9d03-a8f8d00b2dde}
   Folder Axis Control: Id {49ec2768-53b2-482d-b44d-ec52fe555e63}
   Folder Error Checks: Id {dad124df-88d7-4412-bdba-255c48b7272a}
   Folder Exit Checks: Id {866f0ce9-c940-4c68-80f5-47885684bea2}
   Folder HMI updates: Id {df5bfcf9-c740-45ae-b19d-3c3cd0aca00f}
   Folder Init Methods: Id {313976c9-8371-4349-a1d4-ac334e51a051}
   Folder Input Checks: Id {3dff40f9-587b-485b-8ffe-a3d1acaecd62}
   Folder MISC: Id {df8274f9-8bfd-43c2-9dbf-d95ad8873f48}
   Folder Motor Control: Id {4367b06a-8be7-4cee-a828-1c414585ef9d}
   Folder Status Updates: Id {912579cd-d079-4ec8-869a-781310624225}
   Method accelerating_tension: Id {51b0940c-2da9-428b-aa7c-7aa4bc946ef3}
   Method all_check: Id {3616b09d-79ac-4d4e-a9a8-9c800c9db7f0}
   Method count_enabled_motors: Id {4a842378-88e5-40ee-b5f2-32e4ab95fb86}
   Method CYCLIC: Id {66242b1c-4d63-4218-b0e7-5f4fc34ce9db}
   Method decelerating_tension: Id {c76da513-9eeb-4494-921e-e9d30e1467af}
   Method determine_motor_state: Id {e8b4b006-30e0-4934-923d-a97aac10b32d}
   Method estop_routine: Id {e370fdf5-060a-481a-8925-f8c00351b401}
   Method find_eta: Id {85e42879-e4fd-44ad-b45f-475c7a661596}
   Method general_error_check: Id {8ba42383-7e8f-4747-9137-d6b0ee74634e}
   Method general_input_check: Id {a3d14995-b6bb-4412-80c9-b4d7fa9675b0}
   Method get_current_progress: Id {504eb237-53a6-4e39-b7e7-217f0cf72225}
   Method hmi_update: Id {15a1114f-a0f7-4eca-8f18-4cf797395fba}
   Method home: Id {e2c62351-b82f-409f-8c6d-bb5032e701a1}
   Method INIT: Id {a56443b6-9d3c-4e19-bf68-551e95d54fd0}
   Method init_coil_model: Id {90edf354-a001-4a69-9922-1b60f25b1548}
   Method input_update: Id {a62c6a9d-53f4-4e3a-966f-6f249a814bd7}
   Method payoff_input_check: Id {70c3f949-5037-419d-bccb-87705ebd3434}
   Method pickup_input_check: Id {3a472a75-4ad8-4147-bca7-de8a29e62be5}
   Method read_status: Id {c26500a1-9771-4061-a160-1627c7f00ff3}
   Method reset: Id {aef7dc8a-f8b9-41a2-9568-128920b7af80}
   Method set_pos_all: Id {dae62719-33d8-49b6-8821-ff4d77998180}
   Method standstill_tension: Id {2810c0a6-5d8e-4e25-8bef-5c7267116cff}
   Method standstill_tension_check: Id {4514199c-9af5-4a98-ad75-0298298ebf12}
   Method stop_all: Id {91a32785-37fe-490f-8e36-a7fa897334e3}
   Method update_error_status: Id {8a130ded-d455-41f2-ac7c-8c70dbeb7a89}
   Method update_torque: Id {ea80d7c9-b122-46ba-af4e-b3e883f32cba}
   Method update_velocity: Id {e3d6da1b-3c09-4f36-8e11-85f4c14af595}
   Method winding_check: Id {31081dd9-0820-42d0-a9d6-769c3442a1c8}
   Method winding_exit_check: Id {d54735ba-4782-466e-8281-2700698b8cff}
   Method winding_tension: Id {b4e997d8-0092-4fca-a6b8-7c2e056fe739} *)
